Omron CX-Programmer project NewProject (CX-Programmer 9.81)

# PLC NewPLC1: CP2E-N N

## Global symbols (name address type ; comment)
Alternate Alternate

## Program NewProgram1 (cyclic task 0)

### Section Section1

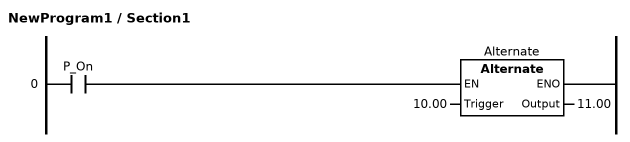
; rung 0
LD P_On
CALL Alternate : Alternate (Trigger := 10.00, Output => 11.00)

### Section END
; rung 0
END(001)

## Function block Alternate
VAR_INPUT
  Trigger : BOOL;
END_VAR
VAR_OUTPUT
  Output : BOOL;
END_VAR
VAR
  Once : BOOL;
END_VAR
IF Trigger AND NOT Once THEN
	Output:= NOT Output;
	Once:=  TRUE;
END_IF;
IF NOT Trigger THEN
	Once :=  FALSE;
END_IF;